// Mitsubishi GX Works2 project: PLC 데이터 명령 (곱셈, 나눗셈)   PLC: Q03UDV

PROGRAM MAIN
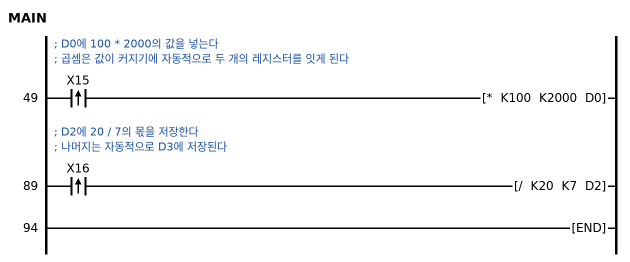
; D0에 100 * 2000의 값을 넣는다
; 곱셈은 값이 커지기에 자동적으로 두 개의 레지스터를 잇게 된다
49    LDP     X15
      *       K100 K2000 D0
; D2에 20 / 7의 몫을 저장한다
; 나머지는 자동적으로 D3에 저장된다
89    LDP     X16
      /       K20 K7 D2
94    END
END_PROGRAM
